{attribute 'linkalways'} 
{attribute 'no_explicit_call' := 'This FB is a CLASS and must be accessed using methods or properties'}
{attribute 'enable_dynamic_creation'}
FUNCTION_BLOCK FINAL Node_DigitalInput EXTENDS HardwareNode
VAR
	input AT %I* : BOOL;
	out : _BOOL(FALSE);
END_VAR

METHOD FB_init : BOOL
VAR_INPUT
	bInitRetains : BOOL; // if TRUE, the retain variables are initialized (warm start / cold start)
	bInCopyCode : BOOL;  // if TRUE, the instance afterwards gets moved into the copy code (online change)
END_VAR
AddOutput('out', out);
END_METHOD

METHOD PROTECTED OnExecute
VAR
END_VAR
out.Value := input;
END_METHOD

END_FUNCTION_BLOCK

(* stored: Version 1.1.0.1, ProductVersion 3.1.4024.13
   POU Node_DigitalInput: Id {0dd4bd2b-0bb5-4458-a128-d5a89ab0178d}, SpecialFunc None
   Folder Constructor: Id {05b25e99-5c4d-4f85-b600-38bc711952f5}
   Method FB_init: Id {d97e36ef-3322-46e9-b125-9ee1f29d291c}
   Method OnExecute: Id {c212795b-274d-4520-8ab4-0c7f2f195a63} *)
